LIN {X 0,Y 56.536,Z 502.549,A -85,B 0,C 180,E1 -30965.975,E2 -30965.975} C_VEL
LIN {X 0,Y 47.794,Z 509.94,A -85,B 0,C 180,E1 -30968.454,E2 -30968.454} C_VEL
LIN {X 0,Y 37.891,Z 516.948,A -85,B 0,C 180,E1 -30973.122,E2 -30973.122} C_VEL
LIN {X 0,Y 29.795,Z 521.793,A -85,B 0,C 180,E1 -30979.326,E2 -30979.326} C_VEL
LIN {X 0,Y 20.85,Z 526.453,A -85,B 0,C 180,E1 -30992.552,E2 -30992.552} C_VEL
LIN {X 0,Y 14.382,Z 529.992,A -85,B 0,C 180,E1 -31020.726,E2 -31020.726} C_VEL
LIN {X 0,Y 13.219,Z 531.761,A -85,B 0,C 180,E1 -31049.981,E2 -31049.981} C_VEL
LIN {X 0,Y 14.432,Z 533.029,A -85,B 0,C 180,E1 -31079.121,E2 -31079.121} C_VEL
LIN {X 0,Y 23.765,Z 534.39,A -85,B 0,C 180,E1 -31112.497,E2 -31112.497} C_VEL
LIN {X 0,Y 29.866,Z 534.466,A -85,B 0,C 180,E1 -31120.241,E2 -31120.241} C_VEL
LIN {X 0,Y 43.03,Z 533.461,A -85,B 0,C 180,E1 -31128.483,E2 -31128.483} C_VEL
LIN {X 0,Y 49.818,Z 532.393,A -85,B 0,C 180,E1 -31130.906,E2 -31130.906} C_VEL
LIN {X 0,Y 57.009,Z 530.819,A -85,B 0,C 180,E1 -31132.92,E2 -31132.92} C_VEL
LIN {X 0,Y 70.501,Z 526.641,A -85,B 0,C 180,E1 -31135.419,E2 -31135.419} C_VEL
LIN {X 0,Y 77.462,Z 523.854,A -85,B 0,C 180,E1 -31136.336,E2 -31136.336} C_VEL
LIN {X 0,Y 81.178,Z 522.113,A -85,B 0,C 180,E1 -31137.136,E2 -31137.136} C_VEL
LIN {X 0,Y 70.291,Z 526.561,A -85,B 0,C 180,E1 -31138.786,E2 -31138.786} C_VEL
LIN {X 0,Y 63.248,Z 528.837,A -85,B 0,C 180,E1 -31140.118,E2 -31140.118} C_VEL
LIN {X 0,Y 56.247,Z 530.663,A -85,B 0,C 180,E1 -31141.784,E2 -31141.784} C_VEL
LIN {X 0,Y 49.303,Z 532.011,A -85,B 0,C 180,E1 -31143.856,E2 -31143.856} C_VEL
LIN {X 0,Y 35.728,Z 533.499,A -85,B 0,C 180,E1 -31150.448,E2 -31150.448} C_VEL
LIN {X 0,Y 29.224,Z 533.629,A -85,B 0,C 180,E1 -31155.886,E2 -31155.886} C_VEL
LIN {X 0,Y 17.697,Z 532.649,A -85,B 0,C 180,E1 -31177.437,E2 -31177.437} C_VEL
LIN {X 0,Y 13.923,Z 531.576,A -85,B 0,C 180,E1 -31199.704,E2 -31199.704} C_VEL
LIN {X 0,Y 15.078,Z 528.6,A -85,B 0,C 180,E1 -31251.2,E2 -31251.2} C_VEL
LIN {X 0,Y 23.143,Z 524.404,A -85,B 0,C 180,E1 -31279.41,E2 -31279.41} C_VEL
LIN {X 0,Y 32.191,Z 519.582,A -85,B 0,C 180,E1 -31290.86,E2 -31290.86} C_VEL
LIN {X 0,Y 41.236,Z 513.953,A -85,B 0,C 180,E1 -31296.979,E2 -31296.979} C_VEL
LIN {X 0,Y 45.641,Z 510.75,A -85,B 0,C 180,E1 -31300.007,E2 -31300.007} C_VEL
LIN {X 0,Y 52.288,Z 505.171,A -85,B 0,C 180,E1 -31305.693,E2 -31305.693} C_VEL
LIN {X 0,Y 58.868,Z 499.041,A -85,B 0,C 180,E1 -31309.983,E2 -31309.983} C_VEL
LIN {X 0,Y 62.92,Z 494.907,A -85,B 0,C 180,E1 -31311.118,E2 -31311.118} C_VEL
LIN {X 0,Y 70.985,Z 485.531,A -85,B 0,C 180,E1 -31311.942,E2 -31311.942} C_VEL
LIN {X 0,Y 78.84,Z 474.119,A -85,B 0,C 180,E1 -31312.642,E2 -31312.642} C_VEL
LIN {X 0,Y 85.484,Z 461.831,A -85,B 0,C 180,E1 -31313.317,E2 -31313.317} C_VEL
LIN {X 0,Y 90.617,Z 449.035,A -85,B 0,C 180,E1 -31313.787,E2 -31313.787} C_VEL
LIN {X 0,Y 94.379,Z 435.682,A -85,B 0,C 180,E1 -31314.126,E2 -31314.126} C_VEL
LIN {X 0,Y 95.113,Z 432.026,A -85,B 0,C 180,E1 -31314.324,E2 -31314.324} C_VEL
LIN {X 0,Y 95.2,Z 431.568,A -85,B 0,C 180,E1 -31315.765,E2 -31315.765} C_VEL
LIN {X 0,Y 95.176,Z 431.749,A -85,B 0,C 180,E1 -31316.194,E2 -31316.194} C_VEL
LIN {X 0,Y 92.024,Z 444.768,A -85,B 0,C 180,E1 -31316.468,E2 -31316.468} C_VEL
LIN {X 0,Y 88.042,Z 456.101,A -85,B 0,C 180,E1 -31316.711,E2 -31316.711} C_VEL
LIN {X 0,Y 82.706,Z 467.537,A -85,B 0,C 180,E1 -31316.885,E2 -31316.885} C_VEL
LIN {X 0,Y 76.53,Z 477.933,A -85,B 0,C 180,E1 -31317.127,E2 -31317.127} C_VEL
LIN {X 0,Y 69.471,Z 487.603,A -85,B 0,C 180,E1 -31317.509,E2 -31317.509} C_VEL
LIN {X 0,Y 61.531,Z 496.573,A -85,B 0,C 180,E1 -31318.173,E2 -31318.173} C_VEL
LIN {X 0,Y 52.72,Z 504.81,A -85,B 0,C 180,E1 -31319.179,E2 -31319.179} C_VEL
LIN {X 0,Y 42.176,Z 512.871,A -85,B 0,C 180,E1 -31320.772,E2 -31320.772} C_VEL
LIN {X 0,Y 31.708,Z 519.342,A -85,B 0,C 180,E1 -31324.021,E2 -31324.021} C_VEL
LIN {X 0,Y 21.39,Z 524.453,A -85,B 0,C 180,E1 -31329.638,E2 -31329.638} C_VEL
LIN {X 0,Y 11.673,Z 528.417,A -85,B 0,C 180,E1 -31345.376,E2 -31345.376} C_VEL
LIN {X 0,Y 6.119,Z 531.318,A -85,B 0,C 180,E1 -31409.958,E2 -31409.958} C_VEL
LIN {X 0,Y 8.928,Z 532.611,A -85,B 0,C 180,E1 -31461.876,E2 -31461.876} C_VEL
LIN {X 0,Y 21.428,Z 534.021,A -85,B 0,C 180,E1 -31489.651,E2 -31489.651} C_VEL
LIN {X 0,Y 28.264,Z 534.145,A -85,B 0,C 180,E1 -31493.963,E2 -31493.963} C_VEL
LIN {X 0,Y 35.207,Z 533.858,A -85,B 0,C 180,E1 -31496.343,E2 -31496.343} C_VEL
LIN {X 0,Y 35.144,Z 533.797,A -85,B 0,C 180,E1 -31498.75,E2 -31498.75} C_VEL
LIN {X 0,Y 28.118,Z 533.972,A -85,B 0,C 180,E1 -31501.583,E2 -31501.583} C_VEL
LIN {X 0,Y 21.194,Z 533.708,A -85,B 0,C 180,E1 -31505.957,E2 -31505.957} C_VEL
LIN {X 0,Y 8.516,Z 532.003,A -85,B 0,C 180,E1 -31534.436,E2 -31534.436} C_VEL
LIN {X 0,Y 6.003,Z 530.543,A -85,B 0,C 180,E1 -31590.042,E2 -31590.042} C_VEL
LIN {X 0,Y 11.546,Z 528.028,A -85,B 0,C 180,E1 -31641.023,E2 -31641.023} C_VEL
LIN {X 0,Y 22.61,Z 523.531,A -85,B 0,C 180,E1 -31658.859,E2 -31658.859} C_VEL
LIN {X 0,Y 34.555,Z 517.359,A -85,B 0,C 180,E1 -31665.066,E2 -31665.066} C_VEL
LIN {X 0,Y 44.894,Z 510.657,A -85,B 0,C 180,E1 -31668.104,E2 -31668.104} C_VEL
LIN {X 0,Y 55.295,Z 502.343,A -85,B 0,C 180,E1 -31670.099,E2 -31670.099} C_VEL
LIN {X 0,Y 62.92,Z 494.907,A -85,B 0,C 180,E1 -31671.118,E2 -31671.118} C_VEL
LIN {X 0,Y 66.345,Z 496.288,A -85,B 0,C 180,E1 -31671.464,E2 -31671.464} C_VEL
LIN {X 0,Y 66.345,Z 600,A -85,B 0,C 180,E1 -31671.464,E2 -31671.464} C_VEL
LIN {X 0,Y 66.345,Z 600,A -85,B 0,C 180,E1 -31671.464,E2 -31671.464}

QRS_NEXT_CUT()

QRS_NEXT()
QRS_HOME()

END
